TYPE ST_ToTc3Hmi_EmergencyStop :
STRUCT
	stName			: ST_Text;
	stItem			: ST_Text;
	nState			: INT;	
END_STRUCT
END_TYPE

(* stored: Version 1.1.0.1, ProductVersion 3.1.4024.11
   DUT ST_ToTc3Hmi_EmergencyStop: Id {3b69382d-5542-4f46-9b18-d0daae2ec689} *)
